(* IEC 61131-3 sources: repolevel_ST_code_completion/real_groud_truth最新/repoeval_Decorator_Application/readful_result, 7 files *)

(* ---- ConcreteComponment.st ---- *)
VAR
    // String field to store the description of the object
    sDescription : STRING;
    // Real field to store the value of the object
    rValue : REAL;
END_VAR

METHOD Initialize : BOOL
VAR_INPUT
    sInitDescription : STRING;
    rInitValue : REAL;
END_VAR
VAR_OUTPUT
END_VAR
VAR
END_VAR

// Method to initialize the ConcreteComponent with a description and value
Initialize := TRUE;
sDescription := sInitDescription;
rValue := rInitValue;

METHOD GetDescription : STRING
VAR_INPUT
END_VAR
VAR_OUTPUT
END_VAR
VAR
END_VAR

// Method to retrieve the description of the component
GetDescription := sDescription;

METHOD GetValue : REAL
VAR_INPUT
END_VAR
VAR_OUTPUT
END_VAR
VAR
END_VAR

// Method to retrieve the value of the component
GetValue := rValue;

METHOD SetDescription : BOOL
VAR_INPUT
    sNewDescription : STRING;
END_VAR
VAR_OUTPUT
END_VAR
VAR
END_VAR

// Method to set a new description for the component
SetDescription := TRUE;
sDescription := sNewDescription;

METHOD SetValue : BOOL
VAR_INPUT
    rNewValue : REAL;
END_VAR
VAR_OUTPUT
END_VAR
VAR
END_VAR

// Method to set a new value for the component
SetValue := TRUE;
rValue := rNewValue;

(* ---- ConcreteComponment_getDescription.st ---- *)
VAR
    // Variable to store the description of the component
    sDescription : STRING;
    // Variable to store the reference to the component being decorated
    tempComponent : Component_Interface;
END_VAR

// Check if the component exists and has a description
IF tempComponent <> NULL THEN
    // Obtain the description of the component and concatenate additional decoration
    getDescription := CONCAT(tempComponent.getDescription(), ' Additional Decoration');
ELSE
    // If no component exists, return a default description
    getDescription := 'Default Description';
END_IF;

(* ---- ConcreteComponment_getValue.st ---- *)
// Assuming this is a continuation of the code structure provided above,
// we will implement the logic for the `getValue` method in a similar manner.

VAR
    // Reference to the component being decorated
    tempComponent : Component_Interface;
    // Additional value for decoration
    decorationValue : REAL := 0.25; // Example decoration value
END_VAR

// Outputs the decorated cost of the component by obtaining the cost of the component to be decorated
// stored in tempComponent.getValue() and then adds the decoration value
getValue := tempComponent.getValue() + decorationValue;

(* ---- ConcreteDecoratorA.st ---- *)
VAR
	//Variable to save the state of the concrete component to be decorated
	tempComponent : Component_Interface;
	//String variable to save the Description of the component
	sDescription : STRING := 'Decorator A';
	//Real variable to save the Value of the component
	rValue : REAL;
END_VAR

METHOD getDescription : STRING
VAR_INPUT
END_VAR

//Outputs the decorated description of the component by obtaining the description of the component
// to be decorated stored in tempComponent.getDescription() and then concatenates the decoration
// description ('Decorator A' as example)
getDescription := CONCAT(THIS^.tempComponent.getDescription(), THIS^.sDescription);

METHOD getValue : REAL
VAR_INPUT
END_VAR

//Outputs the decorated value of the component by obtaining the value of the component
// to be decorated stored in tempComponent.getValue() and then adds the decoration value
getValue := THIS^.tempComponent.getValue() + THIS^.rValue;

(* ---- ConcreteDecoratorA_getDescription.st ---- *)
VAR_OUTPUT
END_VAR
VAR
	//Variable to save the state of the concrete component to be decorated
	tempComponent : Component_Interface;
	//String variable to save the Description of the component
	sDescription : STRING;
	//Real variable to save the Value of the component
	rValue : REAL;
END_VAR

// Check if the input component is valid
IF tempInputComponent <> 0 THEN
	// Assign the input component to the temporary component
	THIS^.tempComponent := tempInputComponent;

	// Concatenate the description of the input component with the decorator's description
	getDescription := CONCAT(THIS^.tempComponent.getDescription(), THIS^.sDescription);
ELSE
	// If no valid input component is provided, return only the decorator's description
	getDescription := THIS^.sDescription;
END_IF;

(* ---- ConcreteDecoratorB.st ---- *)
VAR
	//Variable to save the state of the concrete component to be decorated
	tempComponent : Component_Interface;
	//String variable to save the Description of the component
	sDescription : STRING := ' Decorator B';
	//Real variable to save the Value of the component
	rValue : REAL;
END_VAR

//Method to get the decorated description of the component
METHOD getDescription : STRING
VAR_INPUT
END_VAR

//Outputs the decorated description of the component by obtaining the description of the component
// to be decorated stored in tempComponent.getDescription() and then concatenates the decoration
// description (' Decorator B' as example)
getDescription := CONCAT(THIS^.tempComponent.getDescription(), THIS^.sDescription);

//Method to get the decorated value of the component
METHOD getValue : REAL
VAR_INPUT
END_VAR

//Outputs the decorated value of the component by obtaining the value of the component
// to be decorated stored in tempComponent.getValue() and then adds the decoration value
// (e.g., adding a specific value to the original value)
getValue := THIS^.tempComponent.getValue() + THIS^.rValue;

(* ---- ConcreteDecoratorC.st ---- *)
VAR
	//Variable to save the state of the concrete component to be decorated
	tempComponent : Component_Interface;
	//String variable to save the Description of the component
	sDescription : STRING := ' Decorator C';
	//Real variable to save the Value of the component
	rValue : REAL;
END_VAR

METHOD getDescription : STRING
VAR_INPUT
	//Reference to store the component to be decorated
	tempInputComponent : Component_Interface;
END_VAR

//Outputs the decorated description of the component by obtaining the description of the component
// to be decorated stored in tempComponent.getDescription() and then concatenates the decoration
// description (' Decorator C' as example)
getDescription := CONCAT(THIS^.tempComponent.getDescription(), THIS^.sDescription);

METHOD getValue : REAL
VAR_INPUT
	//Reference to store the component to be decorated
	tempInputComponent : Component_Interface;
END_VAR

//Outputs the decorated value of the component by obtaining the value of the component
// to be decorated stored in tempComponent.getValue() and then adds the decoration value
// (e.g., adding a specific value or applying a transformation)
getValue := THIS^.tempComponent.getValue() + THIS^.rValue;
